(* PLC project SFC_Evolution_1, Beckhoff Automation GmbH TwinCAT PLC Control 3.5.10.30 *)
(* stored: creationDateTime 2019-09-26T15:32:08.5938906, modificationDateTime 2019-09-26T15:32:08.5938906 *)

PROGRAM Main
VAR
	VAR_1: BOOL;
	Condition_1: BOOL;
	Condition_2: BOOL;
END_VAR

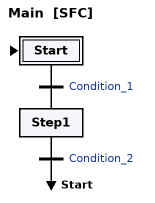
INITIAL_STEP Start:
END_STEP
TRANSITION FROM Start TO Step1
  := Condition_1;
END_TRANSITION
STEP Step1:
END_STEP
TRANSITION FROM Step1 TO Start
  := Condition_2;
END_TRANSITION
END_PROGRAM

CONFIGURATION Application
  RESOURCE SFC_Evolution_1 ON PLC
    TASK PlcTask(INTERVAL := T#0ms, PRIORITY := 20);
    PROGRAM Main WITH PlcTask : Main;
  END_RESOURCE
END_CONFIGURATION
